Universal Robots PolyScope program: Collaboration_Fixture.urp

Program Collaboration_Fixture (installation=Collaboration_Fixture directory=/home/cobot/ursim-5.11.5.1010327/programs createdIn=5.11.5.1010327 lastSavedIn=5.11.5.1010327 robotSerialNumber=20195599999)
Calibrated DH parameters: a=[0, -0.425, -0.3922, 0, 0, 0]; d=[0.1625, 0, 0, 0.1333, 0.0997, 0.0996]; alpha=[1.570796, 0, 0, 1.570796, -1.570796, 0]; deltaTheta=[0, 0, 0, 0, 0, 0]
Robot Program (runOnlyOnce=false)
  Wait DigitalInput pin=ib64; digitalValue=1
  Switch expression=ii24_step
    Case (caseValue=1)
      'Move to Home position'
      SafeHome (positionOptionType=SPEED_AND_ACCELERATION speed=1.047198 acceleration=1.396263 nextMotionTime=2)
    Case (caseValue=2)
      'Move to pickup position and grab a part'
      MoveJ speed 60 deg/s, acceleration 80 deg/s^2 (useActiveTCP=true) feature=Base
        Waypoint Waypoint (Variable): variable(featureName=GrabPosOffset)
      MoveL speed 250 mm/s, acceleration 1200 mm/s^2 (useActiveTCP=true) feature=Base
        Waypoint Waypoint (Variable): variable(featureName=GrabPos)
      Wait Sleep waitTime=2
      MoveL speed 250 mm/s, acceleration 1200 mm/s^2 (useActiveTCP=true) feature=Base
        Waypoint Waypoint (Variable): variable(featureName=GrabPosOffset)
      SafeHome (positionOptionType=SPEED_AND_ACCELERATION speed=1.047198 acceleration=1.396263 nextMotionTime=2)
    Case (caseValue=3)
      'Move to mounting position'
      Switch expression=ii25_actWspace
        Case (caseValue=1)
          MoveJ speed 60 deg/s, acceleration 80 deg/s^2 (useActiveTCP=true) feature=Base
            Waypoint Waypoint (Variable): variable(featureName=MountingTopL)
        Case (caseValue=2)
          MoveJ speed 60 deg/s, acceleration 80 deg/s^2 (useActiveTCP=true) feature=Base
            Waypoint Waypoint (Variable): variable(featureName=MountingTopM)
        Case (caseValue=3)
          MoveJ speed 60 deg/s, acceleration 80 deg/s^2 (useActiveTCP=true) feature=Base
            Waypoint Waypoint (Variable): variable(featureName=MountingTopR)
        Case (caseValue=4)
          MoveJ speed 60 deg/s, acceleration 80 deg/s^2 (useActiveTCP=true) feature=Base
            Waypoint Waypoint (Variable): variable(featureName=MountingBotL)
        Case (caseValue=5)
          MoveJ speed 60 deg/s, acceleration 80 deg/s^2 (useActiveTCP=true) feature=Base
            Waypoint Waypoint (Variable): variable(featureName=MountingBotM)
        Case (caseValue=6)
          MoveJ speed 60 deg/s, acceleration 80 deg/s^2 (useActiveTCP=true) feature=Base
            Waypoint Waypoint (Variable): variable(featureName=MountingBotR)
    Case (caseValue=2147483647)
      'Do nothing (just handshake)'
  Set DigitalOutput pin=ob64; digitalValue=1
  Wait DigitalInput pin=ib64; digitalValue=0
  Set DigitalOutput pin=ob64; digitalValue=0
